// TIA Portal V19 export
FUNCTION_BLOCK "FB10_ManageVacuum"   // FB10, LAD
{ S7_Optimized_Access := 'TRUE' }
// stored: AutoNumber false, IsIECCheckEnabled true, MemoryReserve 100, SetENOAutomatically true
   VAR_INPUT
      xFirstScan { ExternalAccessible := 'False'; ExternalVisible := 'False'; ExternalWritable := 'False'} : Bool;
      xSafetyOk { ExternalAccessible := 'False'; ExternalVisible := 'False'; ExternalWritable := 'False'} : Bool;   // General Safety state
      xAuthorToStart { ExternalAccessible := 'False'; ExternalVisible := 'False'; ExternalWritable := 'False'} : Bool;   // Authorisation to start Vacuum
      xModeAuto { ExternalAccessible := 'False'; ExternalVisible := 'False'; ExternalWritable := 'False'} : Bool;   // Mode auto active
      xResetFault { ExternalAccessible := 'False'; ExternalVisible := 'False'; ExternalWritable := 'False'} : Bool;   // Reset fault
      xBigbagFull { ExternalAccessible := 'False'; ExternalVisible := 'False'; ExternalWritable := 'False'} : Bool;   // Big Bag is full
      xManualReqChangeBigBag { ExternalAccessible := 'False'; ExternalVisible := 'False'; ExternalWritable := 'False'} : Bool;   // Manual request changing Big bag
      xManualStartVacuum { ExternalAccessible := 'False'; ExternalVisible := 'False'; ExternalWritable := 'False'} : Bool;   // Manual enabling Vacuum
      xManualStopVacuum { ExternalAccessible := 'False'; ExternalVisible := 'False'; ExternalWritable := 'False'} : Bool;   // Manual stopping Vacuum
      xLeftRobotReqVacuum { ExternalAccessible := 'False'; ExternalVisible := 'False'; ExternalWritable := 'False'} : Bool;   // Left Robot request enabling Vacuum
      xRightRobotReqVacuum { ExternalAccessible := 'False'; ExternalVisible := 'False'; ExternalWritable := 'False'} : Bool;   // Right Robot request enabling Vacuum
      xVacuumPumpRunning { ExternalAccessible := 'False'; ExternalVisible := 'False'; ExternalWritable := 'False'} : Bool;   // Vacuum Pump Running
      usiActMaterial { ExternalAccessible := 'False'; ExternalVisible := 'False'; ExternalWritable := 'False'} : USInt;   // Type of material for actual production
      xFanDriveRunning { ExternalAccessible := 'False'; ExternalVisible := 'False'; ExternalWritable := 'False'} : Bool;   // State fan drive running
      xFanDriveFault { ExternalAccessible := 'False'; ExternalVisible := 'False'; ExternalWritable := 'False'} : Bool;   // fault fan drive
      xFanFault { ExternalAccessible := 'False'; ExternalVisible := 'False'; ExternalWritable := 'False'} : Bool;   // Fault fan
      xValveMotorFault { ExternalAccessible := 'False'; ExternalVisible := 'False'; ExternalWritable := 'False'} : Bool;   // Fault Valve motor
      xSequencerFault { ExternalAccessible := 'False'; ExternalVisible := 'False'; ExternalWritable := 'False'} : Bool;   // Fault sequencer
   END_VAR
   VAR_OUTPUT
      xStratVacuum { ExternalAccessible := 'False'; ExternalVisible := 'False'; ExternalWritable := 'False'} : Bool;   // Start Vacuum
      xStopVacuum { ExternalAccessible := 'False'; ExternalVisible := 'False'; ExternalWritable := 'False'} : Bool;   // Stop Vacuum
      xBigBagChangeRequest { ExternalAccessible := 'False'; ExternalVisible := 'False'; ExternalWritable := 'False'} : Bool;   // Big Bag change request
      xSandingAuthorization { ExternalAccessible := 'False'; ExternalVisible := 'False'; ExternalWritable := 'False'} : Bool;   // Sanding authorisation
      xFaultActive { ExternalAccessible := 'False'; ExternalVisible := 'False'; ExternalWritable := 'False'} : Bool;
      wVacuumStatus { ExternalAccessible := 'False'; ExternalVisible := 'False'; ExternalWritable := 'False'} : Word;   // Vacuum Status for HMI
      wFault { ExternalAccessible := 'False'; ExternalVisible := 'False'; ExternalWritable := 'False'} : Word;   // Fault number
   END_VAR
   VAR_IN_OUT
      xBigBagChanged { ExternalAccessible := 'False'; ExternalVisible := 'False'; ExternalWritable := 'False'} : Bool;   // Validation operator Big Bag changed
   END_VAR
   VAR
      sxBigBagChangeReq { ExternalAccessible := 'False'; ExternalVisible := 'False'; ExternalWritable := 'False'} : Bool;
      sxVacuumAuto { ExternalAccessible := 'False'; ExternalVisible := 'False'; ExternalWritable := 'False'} : Bool;
      sxVacuumManual { ExternalAccessible := 'False'; ExternalVisible := 'False'; ExternalWritable := 'False'} : Bool;
      sxToggleAuto { ExternalAccessible := 'False'; ExternalVisible := 'False'; ExternalWritable := 'False'} : Bool;
   END_VAR
   VAR RETAIN
      susiPrevMaterial { ExternalAccessible := 'False'; ExternalVisible := 'False'; ExternalWritable := 'False'} : USInt;   // Type of material for previus production
   END_VAR
   VAR
      suiStep { ExternalAccessible := 'False'; ExternalVisible := 'False'; ExternalWritable := 'False'} : UInt;
      miDB_RobotReqVacuum { ExternalAccessible := 'False'; ExternalVisible := 'False'; ExternalWritable := 'False'; S7_SetPoint := 'True'} : TOF_TIME;
      miDB_TonAuthorToStart { ExternalAccessible := 'False'; ExternalVisible := 'False'; ExternalWritable := 'False'; S7_SetPoint := 'True'} : TON_TIME;
      miDB_TonSetp10 { ExternalAccessible := 'False'; ExternalVisible := 'False'; ExternalWritable := 'False'; S7_SetPoint := 'True'} : TON_TIME;
   END_VAR
   VAR CONSTANT
      cuiInitialStep : UInt := 0;
      cuiWaitBigBagChanged : UInt := 5;
      cuiWaitStartVacuum : UInt := 10;
      cuiRunVacuum : UInt := 15;
      cuiWaitStopVacuum : UInt := 20;
      cuiStopVacuum : UInt := 25;
   END_VAR
BEGIN

REGION Network 1 (SCL): Fault number
   // Reset fault
   IF #xResetFault THEN
     #wFault := 16#0;
   END_IF;

   // Sequencer fault
   IF NOT #xSequencerFault THEN
     #wFault.%X0 := TRUE;
   END_IF;

   // Fan drive fault
   IF #xFanDriveFault THEN
     #wFault.%X1 := TRUE;
   END_IF;

   // Breaker 11Q1 in AER cabinet fault
   IF #xFanFault AND (NOT #xFanDriveFault) THEN
     #wFault.%X2 := TRUE;
   END_IF;

   // Breaker 10Q1 in AER cabinet fault
   IF #xValveMotorFault THEN
     #wFault.%X3 := TRUE;
   END_IF;

   #miDB_TonAuthorToStart(IN:=(NOT #xFanDriveRunning) AND (NOT #xAuthorToStart),
                          PT:=T#10S);
   IF #miDB_TonAuthorToStart.Q THEN
     #wFault.%X4 := TRUE;
   END_IF;

   // At least one active fault
   #xFaultActive := (#wFault <> 16#0);
END_REGION

REGION Network 2: At least one robot request vacumm
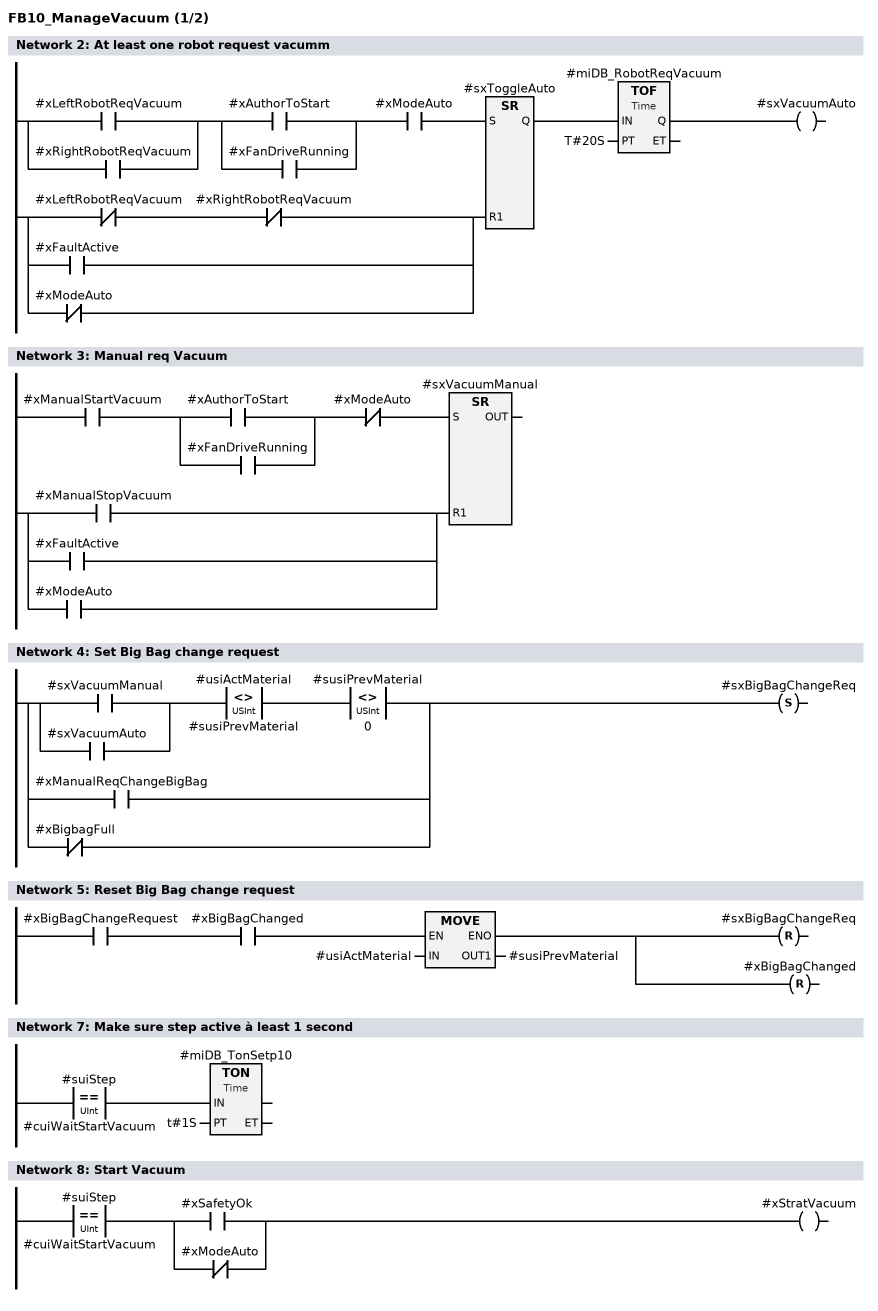
   RUNG wire#powerrail
      Contact( #xLeftRobotReqVacuum )
      wire#w1
      Contact( #xAuthorToStart )
      wire#w2
      Contact( #xModeAuto )
      S_SR(operand := #sxToggleAuto, r1 := wire#w3)
      { S7_Templates := "time_type := Time" } #miDB_RobotReqVacuum.TOF(pt := T#20S, et =>)
      Coil( #sxVacuumAuto )
   END_RUNG
   RUNG wire#powerrail
      Contact( #xRightRobotReqVacuum )
   END_RUNG wire#w1
   RUNG wire#w1
      Contact( #xFanDriveRunning )
   END_RUNG wire#w2
   RUNG wire#powerrail
      I_Contact( #xLeftRobotReqVacuum )
      I_Contact( #xRightRobotReqVacuum )
   END_RUNG wire#w3
   RUNG wire#powerrail
      Contact( #xFaultActive )
   END_RUNG wire#w3
   RUNG wire#powerrail
      I_Contact( #xModeAuto )
   END_RUNG wire#w3
   // the same network as SCL:
   IF (#xLeftRobotReqVacuum OR #xRightRobotReqVacuum) AND (#xAuthorToStart OR #xFanDriveRunning) AND #xModeAuto THEN
       #sxToggleAuto := TRUE;   // SR flip-flop
   END_IF;
   IF (NOT #xLeftRobotReqVacuum AND NOT #xRightRobotReqVacuum) OR #xFaultActive OR NOT #xModeAuto THEN
       #sxToggleAuto := FALSE;
   END_IF;
   #miDB_RobotReqVacuum(IN := #sxToggleAuto, PT := T#20S);   // TOF
   #sxVacuumAuto := #miDB_RobotReqVacuum.Q;
END_REGION

REGION Network 3: Manual req Vacuum
   RUNG wire#powerrail
      Contact( #xManualStartVacuum )
      wire#w1
      Contact( #xAuthorToStart )
      wire#w2
      I_Contact( #xModeAuto )
      S_SR(operand := #sxVacuumManual, r1 := wire#w3)
   END_RUNG
   RUNG wire#w1
      Contact( #xFanDriveRunning )
   END_RUNG wire#w2
   RUNG wire#powerrail
      Contact( #xManualStopVacuum )
   END_RUNG wire#w3
   RUNG wire#powerrail
      Contact( #xFaultActive )
   END_RUNG wire#w3
   RUNG wire#powerrail
      Contact( #xModeAuto )
   END_RUNG wire#w3
   // the same network as SCL:
   IF #xManualStartVacuum AND (#xAuthorToStart OR #xFanDriveRunning) AND NOT #xModeAuto THEN
       #sxVacuumManual := TRUE;   // SR flip-flop
   END_IF;
   IF #xManualStopVacuum OR #xFaultActive OR #xModeAuto THEN #sxVacuumManual := FALSE; END_IF;
END_REGION

REGION Network 4: Set Big Bag change request
   RUNG wire#powerrail
      Contact( #sxVacuumManual )
      wire#w1
      { S7_Templates := "SrcType := USInt" } NE_Contact(in1 := #usiActMaterial, in2 := #susiPrevMaterial)
      { S7_Templates := "SrcType := USInt" } NE_Contact(in1 := #susiPrevMaterial, in2 := 0)
      wire#w2
      S_Coil( #sxBigBagChangeReq )
   END_RUNG
   RUNG wire#powerrail
      Contact( #sxVacuumAuto )
   END_RUNG wire#w1
   RUNG wire#powerrail
      Contact( #xManualReqChangeBigBag )
   END_RUNG wire#w2
   RUNG wire#powerrail
      I_Contact( #xBigbagFull )
   END_RUNG wire#w2
   // the same network as SCL:
   IF ((#sxVacuumManual OR #sxVacuumAuto) AND (#usiActMaterial <> #susiPrevMaterial) AND (#susiPrevMaterial <> 0)) OR #xManualReqChangeBigBag OR NOT #xBigbagFull THEN
       #sxBigBagChangeReq := TRUE;
   END_IF;
END_REGION

REGION Network 5: Reset Big Bag change request
   RUNG wire#powerrail
      Contact( #xBigBagChangeRequest )
      Contact( #xBigBagChanged )
      Move(in := #usiActMaterial, out1 => #susiPrevMaterial)
      wire#w1
      R_Coil( #sxBigBagChangeReq )
   END_RUNG
   RUNG wire#w1
      R_Coil( #xBigBagChanged )
   END_RUNG
   // the same network as SCL:
   IF #xBigBagChangeRequest AND #xBigBagChanged THEN
       #susiPrevMaterial := #usiActMaterial;
       #sxBigBagChangeReq := FALSE;
       #xBigBagChanged := FALSE;
   END_IF;
END_REGION

REGION Network 6 (SCL): Sequencer Vacuum
   // Initialise sequence at first scan of PLC
   IF #xFirstScan THEN
     #suiStep := #cuiInitialStep;
   END_IF;

   // Sequencer step
   CASE #suiStep OF
     #cuiInitialStep:
       IF (#sxVacuumAuto OR #sxVacuumManual) AND #xSafetyOk AND (NOT #sxBigBagChangeReq) THEN
         #suiStep := #cuiWaitStartVacuum;
       ELSIF (#sxVacuumAuto OR #sxVacuumManual) AND #xSafetyOk AND #sxBigBagChangeReq THEN
         #suiStep := #cuiWaitBigBagChanged;
       END_IF;

     #cuiWaitBigBagChanged:
       IF (NOT #sxBigBagChangeReq) THEN
         #suiStep := #cuiWaitStartVacuum;
       END_IF;

     #cuiWaitStartVacuum:
       IF #xFanDriveRunning AND #miDB_TonSetp10.Q THEN
         #suiStep := #cuiRunVacuum;
       END_IF;

     #cuiRunVacuum:
       IF ((NOT #sxVacuumAuto) AND (NOT #sxVacuumManual)) OR (NOT #xSafetyOk) THEN
         #suiStep := #cuiWaitStopVacuum;
       END_IF;

     #cuiWaitStopVacuum:
       IF (NOT #xFanDriveRunning) THEN
         #suiStep := #cuiStopVacuum;
       ELSIF (#sxVacuumAuto OR #sxVacuumManual) AND #xSafetyOk THEN
         #suiStep := #cuiWaitStartVacuum;
       END_IF;

     #cuiStopVacuum:
       IF #xAuthorToStart THEN;
         #suiStep := #cuiInitialStep;
       END_IF;

     ELSE  // Statement section ELSE
       // Error in this case
       ;
   END_CASE;
END_REGION

REGION Network 7: Make sure step active à least 1 second
   RUNG wire#powerrail
      { S7_Templates := "SrcType := UInt" } EQ_Contact(in1 := #suiStep, in2 := #cuiWaitStartVacuum)
      { S7_Templates := "time_type := Time" } #miDB_TonSetp10.TON(pt := t#1S, et =>)
   END_RUNG
   // the same network as SCL:
   #miDB_TonSetp10(IN := #suiStep = #cuiWaitStartVacuum, PT := t#1S);   // TON
END_REGION

REGION Network 8: Start Vacuum
   RUNG wire#powerrail
      { S7_Templates := "SrcType := UInt" } EQ_Contact(in1 := #suiStep, in2 := #cuiWaitStartVacuum)
      wire#w1
      Contact( #xSafetyOk )
      wire#w2
      Coil( #xStratVacuum )
   END_RUNG
   RUNG wire#w1
      I_Contact( #xModeAuto )
   END_RUNG wire#w2
   // the same network as SCL:
   #xStratVacuum := (#suiStep = #cuiWaitStartVacuum) AND (#xSafetyOk OR NOT #xModeAuto);
END_REGION

REGION Network 9: Stop Vacuum
   // Shunt a enlever
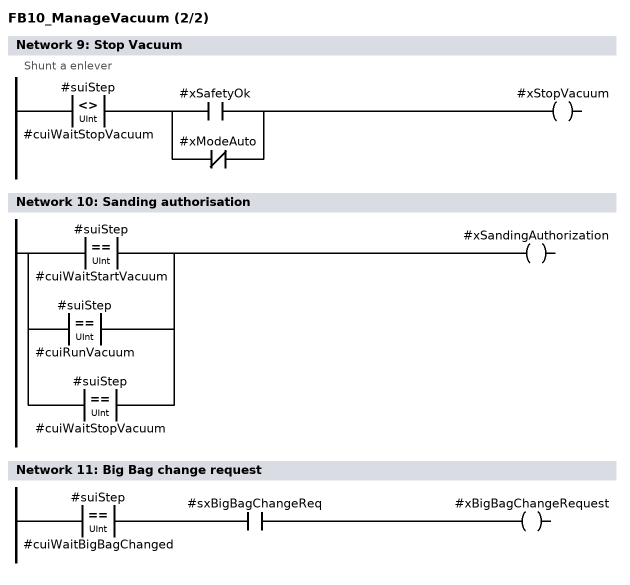
   RUNG wire#powerrail
      { S7_Templates := "SrcType := UInt" } NE_Contact(in1 := #suiStep, in2 := #cuiWaitStopVacuum)
      wire#w1
      Contact( #xSafetyOk )
      wire#w2
      Coil( #xStopVacuum )
   END_RUNG
   RUNG wire#w1
      I_Contact( #xModeAuto )
   END_RUNG wire#w2
   // the same network as SCL:
   #xStopVacuum := (#suiStep <> #cuiWaitStopVacuum) AND (#xSafetyOk OR NOT #xModeAuto);
END_REGION

REGION Network 10: Sanding authorisation
   RUNG wire#powerrail
      { S7_Templates := "SrcType := UInt" } EQ_Contact(in1 := #suiStep, in2 := #cuiWaitStartVacuum)
      wire#w1
      Coil( #xSandingAuthorization )
   END_RUNG
   RUNG wire#powerrail
      { S7_Templates := "SrcType := UInt" } EQ_Contact(in1 := #suiStep, in2 := #cuiRunVacuum)
   END_RUNG wire#w1
   RUNG wire#powerrail
      { S7_Templates := "SrcType := UInt" } EQ_Contact(in1 := #suiStep, in2 := #cuiWaitStopVacuum)
   END_RUNG wire#w1
   // the same network as SCL:
   #xSandingAuthorization := (#suiStep = #cuiWaitStartVacuum) OR (#suiStep = #cuiRunVacuum) OR (#suiStep = #cuiWaitStopVacuum);
END_REGION

REGION Network 11: Big Bag change request
   RUNG wire#powerrail
      { S7_Templates := "SrcType := UInt" } EQ_Contact(in1 := #suiStep, in2 := #cuiWaitBigBagChanged)
      Contact( #sxBigBagChangeReq )
      Coil( #xBigBagChangeRequest )
   END_RUNG
   // the same network as SCL:
   #xBigBagChangeRequest := (#suiStep = #cuiWaitBigBagChanged) AND #sxBigBagChangeReq;
END_REGION

REGION Network 12 (SCL): Vacuum Status
   // Reset Vacuum Status
   #wVacuumStatus := 16#0;
   // If Fault set bit 1
   IF #xFaultActive THEN // Show at list one fault active
     #wVacuumStatus := 16#1;
   ELSIF (NOT #xBigbagFull) THEN // Big Bag Full
     #wVacuumStatus := 16#2;
   ELSE
     // Fan drive activated
     IF #xFanDriveRunning THEN
       #wVacuumStatus := #wVacuumStatus OR 16#4;
     END_IF;

     // VacuumPump running
     IF #xVacuumPumpRunning THEN
       #wVacuumStatus := #wVacuumStatus OR 16#8;
     END_IF;

     CASE #suiStep OF

       #cuiInitialStep:
         #wVacuumStatus := #wVacuumStatus OR 16#10;

       #cuiWaitBigBagChanged:
         #wVacuumStatus := #wVacuumStatus OR 16#20;

       #cuiWaitStartVacuum, #cuiRunVacuum:
         #wVacuumStatus := #wVacuumStatus OR 16#40;

       #cuiWaitStopVacuum, #cuiStopVacuum:
         #wVacuumStatus := #wVacuumStatus OR 16#80;

     END_CASE;
   END_IF;
END_REGION
END_FUNCTION_BLOCK
